FUNCTION F_Convert_Uint_to_2Byte
VAR_IN_OUT
	inputNum : UINT; 
	dataByte1 : BYTE;
	dataByte2 : BYTE;
END_VAR

VAR
	arrByte : ARRAY [0..1] OF BYTE;
END_VAR

MEMCPY(ADR(arrByte), ADR(inputNum), 2);
dataByte1 := arrByte[0];
dataByte2 := arrByte[1];

//F_Convert_Int_to_2Byte:=arrByte;

END_FUNCTION

(* stored: Version 1.1.0.1, ProductVersion 3.1.4024.11
   POU F_Convert_Uint_to_2Byte: Id {8efc81d2-ee47-47d4-8f53-c81d38f0bed8}, SpecialFunc None *)
